Fanuc TP program (LS listing): UP206.LS

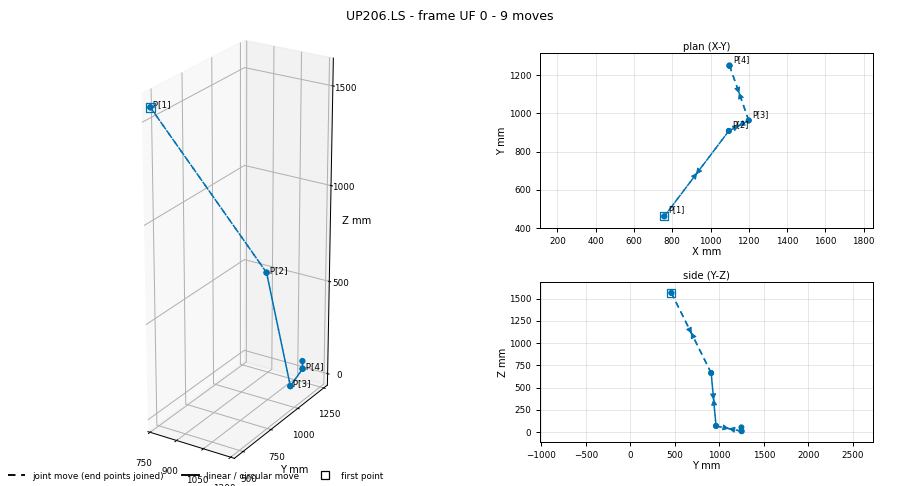
[picture p0: tool path of UP206.LS in frame UF 0, 9 of 9 moves have a stored position in this frame; points joined in program order, loops and branches not executed]
/PROG  UP206
/ATTR
OWNER		= SHIFT;
COMMENT		= "Prueba TCP SP1";
PROG_SIZE	= 3492;
CREATE		= DATE 16-10-11  TIME 22:47:06;
MODIFIED	= DATE 17-06-27  TIME 08:39:10;
FILE_NAME	= UP209;
VERSION		= 0;
LINE_COUNT	= 16;
MEMORY_SIZE	= 7100;
PROTECT		= READ_WRITE;
TCD:  STACK_SIZE	= 500,
      TASK_PRIORITY	= 50,
      TIME_SLICE	= 0,
      BUSY_LAMP_OFF	= 0,
      ABORT_REQUEST	= 0,
      PAUSE_REQUEST	= 0;
DEFAULT_GROUP	= 1,1,1,1,*;
CONTROL_CODE	= 00000000 00000000;
/APPL
/MN
   1:  UTOOL_NUM=24 ;
   2:  UFRAME_NUM=0 ;
   3:  PAYLOAD[1] ;
   4:J P[1] 100% CNT0 ACC100 TB    .10sec,P-SPS    ;
      1:  TC_ONLINE (ON) ;
      2:  DO[23]=OFF ;
      3:  CALL MAKRO050    ;
      4:  WAIT (DO[11])    ;
      5:  WAIT (DI[23])    ;
      6:  DO[23]=ON ;
      7:  TC_ONLINE (M[30] AND M[95]) ;
       ------ ;
   5:J P[2] 100% CNT100 ACC100 TB   0.00sec,P-SPS    ;
      1:  TC_ONLINE (M[30] AND M[95]) ;
       ------ ;
   6:J P[3] 100% CNT100 ACC100 TB   0.00sec,P-SPS    ;
      1:  TC_ONLINE (M[30] AND M[95]) ;
       ------ ;
   7:J P[4] 100% CNT0 ACC100 TB    .10sec,P-SPS    ;
      1:  TC_ONLINE (ON) ;
      2:  DO[23]=OFF ;
      3:  WAIT (DI[23])    ;
      4:  DO[23]=ON ;
      5:  TC_ONLINE (M[30] AND M[95]) ;
       ------ ;
   8:  !Posicion Prueba TCP ;
   9:  !SP1 ;
  10:  !X=1099.530 Y=1249.375 Z=54.007 ;
  11:  !W=-18.409 P=-89.280 R=-52.358 ;
  12:L P[5] 400mm/sec CNT0 ACC100 TB    .10sec,P-SPS    ;
      1:  TC_ONLINE (ON) ;
      2:  DO[23]=OFF ;
      3:  WAIT (DI[17])    ;
      4:  WAIT (DI[23])    ;
      5:  DO[23]=ON ;
      6:  TC_ONLINE (M[30] AND M[95]) ;
       ------ ;
  13:L P[6] 400mm/sec CNT0 ACC100 TB    .10sec,P-SPS    ;
      1:  TC_ONLINE (ON) ;
      2:  DO[23]=OFF ;
      3:  WAIT (DI[23])    ;
      4:  DO[23]=ON ;
      5:  TC_ONLINE (M[30] AND M[95]) ;
       ------ ;
  14:J P[7] 100% CNT100 ACC100 TB   0.00sec,P-SPS    ;
      1:  TC_ONLINE (M[30] AND M[95]) ;
       ------ ;
  15:J P[8] 100% CNT100 ACC100 TB   0.00sec,P-SPS    ;
      1:  TC_ONLINE (M[30] AND M[95]) ;
       ------ ;
  16:J P[9] 100% CNT0 ACC100 TB    .10sec,P-SPS    ;
      1:  TC_ONLINE (ON) ;
      2:  DO[23]=OFF ;
      3:  WAIT (DI[23])    ;
      4:  DO[23]=ON ;
      5:  TC_ONLINE (M[30] AND M[95]) ;
       ------ ;
/POS
P[1]{
   GP1:
	UF : 0, UT : 24,		CONFIG : 'N U T, 0, 0, 0',
	X =   758.413  mm,	Y =   461.520  mm,	Z =  1563.091  mm,
	W =  -172.162 deg,	P =   -29.440 deg,	R =    24.278 deg
   GP2:
	UF : 0, UT : 24,
	J1=   100.000  mm
   GP3:
	UF : 0, UT : 24,
	J1=     0.000  mm
   GP4:
	UF : 0, UT : 24,
	J1=     0.000  mm
};
P[2]{
   GP1:
	UF : 0, UT : 24,		CONFIG : 'N U T, 0, 0, 0',
	X =  1095.863  mm,	Y =   908.045  mm,	Z =   663.757  mm,
	W =  -157.913 deg,	P =   -55.962 deg,	R =    79.866 deg
   GP2:
	UF : 0, UT : 24,
	J1=   100.000  mm
   GP3:
	UF : 0, UT : 24,
	J1=     0.000  mm
   GP4:
	UF : 0, UT : 24,
	J1=     0.000  mm
};
P[3]{
   GP1:
	UF : 0, UT : 24,		CONFIG : 'N U T, 0, 0, 0',
	X =  1199.720  mm,	Y =   962.639  mm,	Z =    68.949  mm,
	W =   -18.400 deg,	P =   -89.280 deg,	R =   -52.353 deg
   GP2:
	UF : 0, UT : 24,
	J1=   100.000  mm
   GP3:
	UF : 0, UT : 24,
	J1=     0.000  mm
   GP4:
	UF : 0, UT : 24,
	J1=     0.000  mm
};
P[4]{
   GP1:
	UF : 0, UT : 24,		CONFIG : 'N U T, 0, 0, 0',
	X =  1099.191  mm,	Y =  1249.813  mm,	Z =     9.932  mm,
	W =   -18.405 deg,	P =   -89.280 deg,	R =   -52.347 deg
   GP2:
	UF : 0, UT : 24,
	J1=   100.000  mm
   GP3:
	UF : 0, UT : 24,
	J1=     0.000  mm
   GP4:
	UF : 0, UT : 24,
	J1=     0.000  mm
};
P[5]{
   GP1:
	UF : 0, UT : 24,		CONFIG : 'N U T, 0, 0, 0',
	X =  1099.024  mm,	Y =  1247.628  mm,	Z =    53.832  mm,
	W =   -19.024 deg,	P =   -89.281 deg,	R =   -51.725 deg
   GP2:
	UF : 0, UT : 24,
	J1=    99.800  mm
   GP3:
	UF : 0, UT : 24,
	J1=     0.000  mm
   GP4:
	UF : 0, UT : 24,
	J1=     0.000  mm
};
P[6]{
   GP1:
	UF : 0, UT : 24,		CONFIG : 'N U T, 0, 0, 0',
	X =  1099.191  mm,	Y =  1249.813  mm,	Z =     9.932  mm,
	W =   -18.405 deg,	P =   -89.280 deg,	R =   -52.347 deg
   GP2:
	UF : 0, UT : 24,
	J1=   100.000  mm
   GP3:
	UF : 0, UT : 24,
	J1=     0.000  mm
   GP4:
	UF : 0, UT : 24,
	J1=     0.000  mm
};
P[7]{
   GP1:
	UF : 0, UT : 24,		CONFIG : 'N U T, 0, 0, 0',
	X =  1199.720  mm,	Y =   962.639  mm,	Z =    68.949  mm,
	W =   -18.400 deg,	P =   -89.280 deg,	R =   -52.353 deg
   GP2:
	UF : 0, UT : 24,
	J1=   100.000  mm
   GP3:
	UF : 0, UT : 24,
	J1=     0.000  mm
   GP4:
	UF : 0, UT : 24,
	J1=     0.000  mm
};
P[8]{
   GP1:
	UF : 0, UT : 24,		CONFIG : 'N U T, 0, 0, 0',
	X =  1095.863  mm,	Y =   908.045  mm,	Z =   663.757  mm,
	W =  -157.913 deg,	P =   -55.962 deg,	R =    79.866 deg
   GP2:
	UF : 0, UT : 24,
	J1=   100.000  mm
   GP3:
	UF : 0, UT : 24,
	J1=     0.000  mm
   GP4:
	UF : 0, UT : 24,
	J1=     0.000  mm
};
P[9]{
   GP1:
	UF : 0, UT : 24,		CONFIG : 'N U T, 0, 0, 0',
	X =   758.413  mm,	Y =   461.520  mm,	Z =  1563.091  mm,
	W =  -172.162 deg,	P =   -29.440 deg,	R =    24.278 deg
   GP2:
	UF : 0, UT : 24,
	J1=   100.000  mm
   GP3:
	UF : 0, UT : 24,
	J1=     0.000  mm
   GP4:
	UF : 0, UT : 24,
	J1=     0.000  mm
};
/END
